PROGRAM P_InitOnce
VAR
	done : BOOL;
	
END_VAR

GVL.firstCycle := FALSE;

IF done THEN
	RETURN;
END_IF

done := TRUE;

GVL.firstCycle := TRUE;


GVL.devSortierer.wID := 100;
GVL.devSortierer.sDevName := 'Sortierer';
GVL.devSortierer.rIN_LO := 0;
GVL.devSortierer.rIN_HI := 100; //ToDo: Checken
GVL.devSortierer.nOUT_LO := 819;
GVL.devSortierer.nOUT_HI := 65535;
GVL.calcDev(Dev := ADR(GVL.devSortierer));

GVL.devDruckVentil.wID := 101;
GVL.devDruckVentil.sDevName := 'Druck-Ventil';
GVL.devDruckVentil.rIN_LO := 0.0;
GVL.devDruckVentil.rIN_HI := 100.0;
GVL.devDruckVentil.nOUT_LO := 0;
GVL.devDruckVentil.nOUT_HI := 65535;
GVL.calcDev(Dev := ADR(GVL.devDruckVentil));


VAT.byBlinkTakt := 0;

DB6.runTime.seconds := 0;

//Später wieder raus
VAT.bSammelStoerung := 0;

RVL.currLogLevel := 8;

DB6.nAusstossverz := REAL_TO_INT(DB6.rAusstossverz * 1000);

MAIN.M_Log(reqLevel:=CVL.INFO, objectName:= 'P_InitOnce', sMsg:='done', errNo:= 0);

IO.safetyRUN := TRUE;

END_PROGRAM

(* stored: Version 1.1.0.1, ProductVersion 3.1.4024.3
   POU P_InitOnce: Id {dd986b0e-7367-479a-a1bc-68a8fa7a387e}, SpecialFunc None *)
